INTERFACE ITF_TopElement2_HMI_Connector_View EXTENDS ITF_BaseTopElement_HMI_Connector_View

END_INTERFACE

(* stored: Version 1.1.0.1
   Itf ITF_TopElement2_HMI_Connector_View: Id {f3ec4c0d-8417-0b5a-3584-2d9c88604c8d} *)
